{attribute 'qualified_only'}
VAR_GLOBAL
END_VAR

(* stored: Version 1.1.0.1
   GVL GVL: Id {423cc0c7-9346-40f2-8bb7-f68480a13c29} *)
